FUNCTION_BLOCK basicRevezamento3Motores (* Basic Function Block Type *)
  (* Standard: 61499-2 *)
  (* Version 0.0, 2/10/2026, Schneider Electric, Template *)
  PACKAGE Hidryco.HidrycoLib;
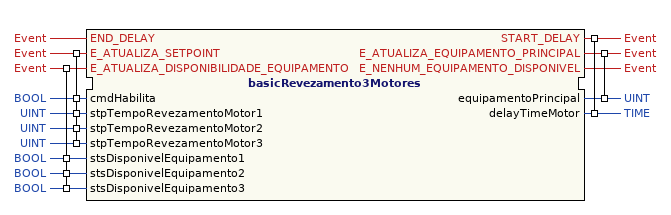
  EVENT_INPUT
    END_DELAY;
    E_ATUALIZA_SETPOINT WITH stpTempoRevezamentoMotor1, stpTempoRevezamentoMotor2, stpTempoRevezamentoMotor3, cmdHabilita;
    E_ATUALIZA_DISPONIBILIDADE_EQUIPAMENTO WITH stsDisponivelEquipamento1, stsDisponivelEquipamento2, stsDisponivelEquipamento3;
  END_EVENT
  EVENT_OUTPUT
    START_DELAY WITH delayTimeMotor;
    E_ATUALIZA_EQUIPAMENTO_PRINCIPAL WITH equipamentoPrincipal;
    E_NENHUM_EQUIPAMENTO_DISPONIVEL;
  END_EVENT
  VAR_INPUT
    cmdHabilita : BOOL;
    stpTempoRevezamentoMotor1 : UINT;
    stpTempoRevezamentoMotor2 : UINT;
    stpTempoRevezamentoMotor3 : UINT;
    stsDisponivelEquipamento1 : BOOL;
    stsDisponivelEquipamento2 : BOOL;
    stsDisponivelEquipamento3 : BOOL;
  END_VAR
  VAR_OUTPUT
    equipamentoPrincipal : UINT := 1;
    delayTimeMotor : TIME;
  END_VAR
  VAR
    equipamentosDisponiveis : INT;
  END_VAR
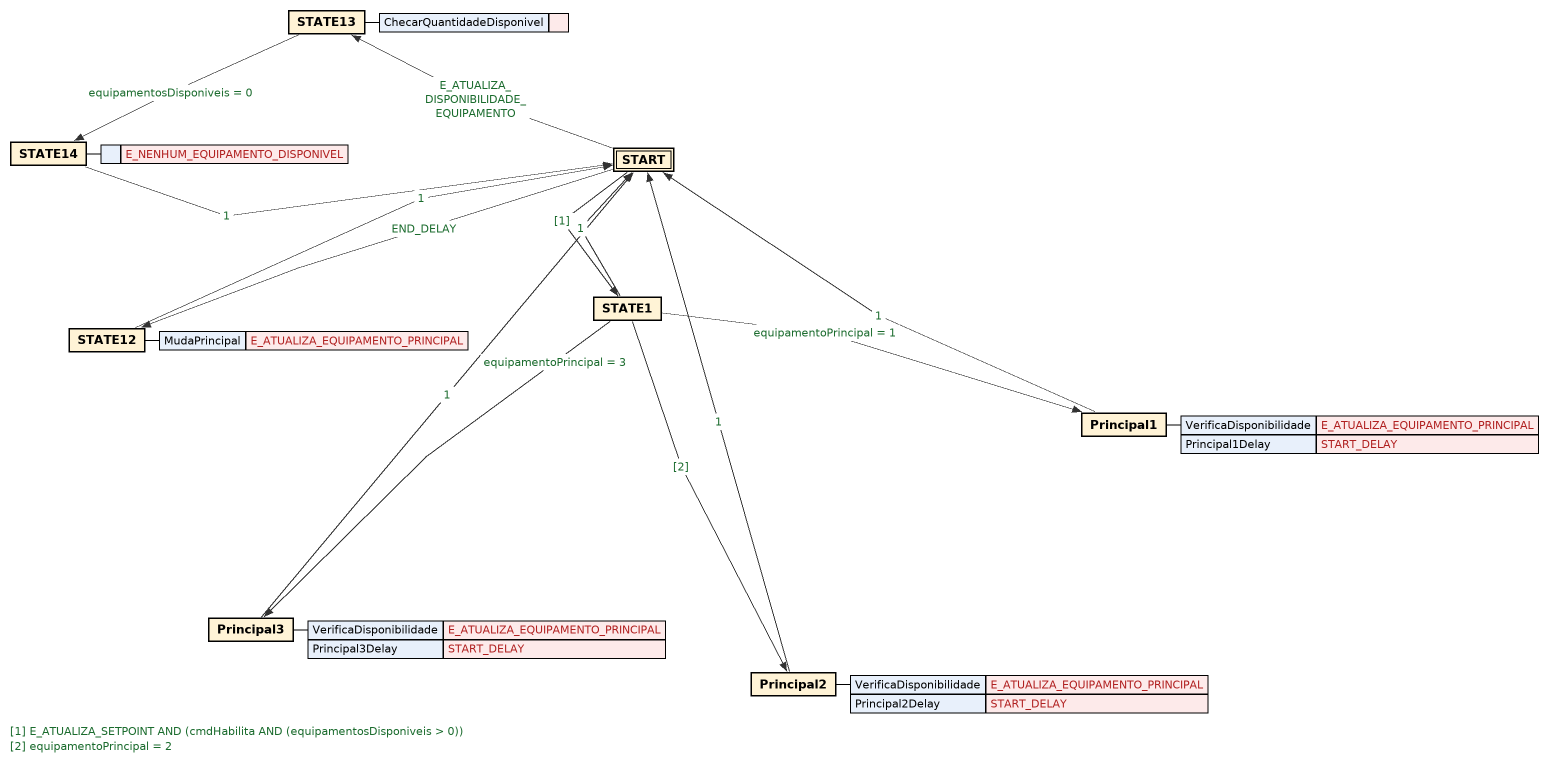
  EC_STATES
    START; (* Initial State *)
    STATE1;
    Principal1 : VerificaDisponibilidade -> E_ATUALIZA_EQUIPAMENTO_PRINCIPAL, Principal1Delay -> START_DELAY;
    Principal2 : VerificaDisponibilidade -> E_ATUALIZA_EQUIPAMENTO_PRINCIPAL, Principal2Delay -> START_DELAY;
    Principal3 : VerificaDisponibilidade -> E_ATUALIZA_EQUIPAMENTO_PRINCIPAL, Principal3Delay -> START_DELAY;
    STATE12 : MudaPrincipal -> E_ATUALIZA_EQUIPAMENTO_PRINCIPAL;
    STATE13 : ChecarQuantidadeDisponivel;
    STATE14 : -> E_NENHUM_EQUIPAMENTO_DISPONIVEL;
  END_STATES
  EC_TRANSITIONS
    START TO STATE13 := E_ATUALIZA_DISPONIBILIDADE_EQUIPAMENTO;
    STATE13 TO STATE14 := equipamentosDisponiveis = 0;
    STATE14 TO START := 1;
    START TO STATE12 := END_DELAY;
    STATE12 TO START := 1;
    START TO STATE1 := E_ATUALIZA_SETPOINT AND (cmdHabilita AND (equipamentosDisponiveis > 0));
    STATE1 TO Principal1 := equipamentoPrincipal = 1;
    Principal1 TO START := 1;
    STATE1 TO Principal2 := equipamentoPrincipal = 2;
    Principal2 TO START := 1;
    STATE1 TO Principal3 := equipamentoPrincipal = 3;
    Principal3 TO START := 1;
    STATE1 TO START := 1;
  END_TRANSITIONS
  ALGORITHM Principal1Delay IN ST:
delayTimeMotor := DINT_TO_TIME(UINT_TO_DINT(stpTempoRevezamentoMotor1)*3600000);
;
  END_ALGORITHM
  ALGORITHM Principal2Delay IN ST:
delayTimeMotor := DINT_TO_TIME(UINT_TO_DINT(stpTempoRevezamentoMotor2)*3600000);
;
  END_ALGORITHM
  ALGORITHM Principal3Delay IN ST:
delayTimeMotor := DINT_TO_TIME(UINT_TO_DINT(stpTempoRevezamentoMotor3)*3600000);
;
  END_ALGORITHM
  ALGORITHM MudaPrincipal IN ST:
IF equipamentoPrincipal > 0 AND equipamentoPrincipal < 3 THEN
	equipamentoPrincipal := equipamentoPrincipal + 1;
ELSE
	equipamentoPrincipal := 1;
END_IF;
;
  END_ALGORITHM
  ALGORITHM ChecarQuantidadeDisponivel IN ST:
equipamentosDisponiveis := BOOL_TO_INT(stsDisponivelEquipamento1) + BOOL_TO_INT(stsDisponivelEquipamento2) +  BOOL_TO_INT(stsDisponivelEquipamento3);
;
  END_ALGORITHM
  ALGORITHM VerificaDisponibilidade IN ST:
IF equipamentoPrincipal = 1 AND NOT stsDisponivelEquipamento1 THEN
	equipamentoPrincipal := equipamentoPrincipal + 1;
ELSIF equipamentoPrincipal = 2 AND NOT stsDisponivelEquipamento2 THEN
	equipamentoPrincipal := equipamentoPrincipal + 1;
ELSIF equipamentoPrincipal = 3 AND NOT stsDisponivelEquipamento3 THEN
	equipamentoPrincipal := 1;
END_IF;
;
  END_ALGORITHM
END_FUNCTION_BLOCK
